{attribute 'qualified_only'}
{attribute 'strict'}
TYPE E_ServoVise_Command :
(
	NoCommand,
	Open,
	Close
);
END_TYPE

(* stored: Version 1.1.0.1, ProductVersion 3.1.4024.11
   DUT E_ServoVise_Command: Id {6d567d06-f76c-480a-9878-61fbe11a8111} *)
